RoboDK station: Model of an industrial robot with a technical vision system for palletizing objects in the RoboDK environment.rdk

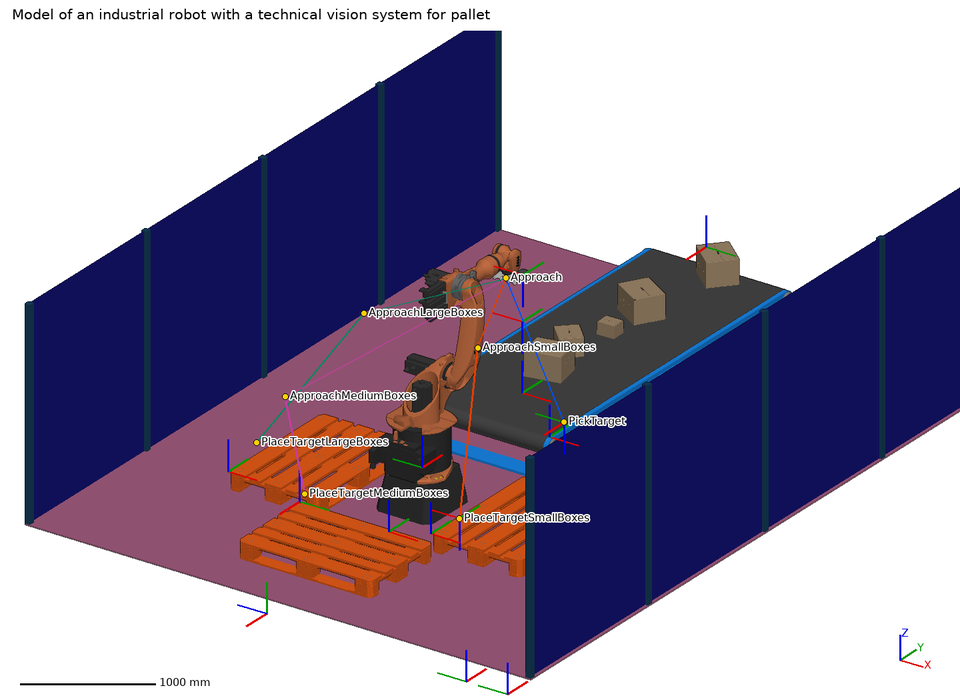
[picture v0: the station drawn from its stored meshes, robots at their saved joint values, targets as dots, program paths as lines]
Station Model of an industrial robot with a technical vision system for palletizing objects in the RoboDK environment (saved by RoboDK 5.9.0). Poses are relative to the parent item; angles as X-Y-Z fixed-axis rotations.
Station parameters (name, value as stored): BOXSPAWNER_SIZE_X, 400.0, BOXSPAWNER_SIZE_Y, 200.0, BOXSPAWNER_SIZE_Z, 200.0, BOXSPAWNER_UNITS, True, BOXSPAWNER_PARENT, Frame 6, BOXSPAWNER_CONV_PARENT, Frame 6, BOXSPAWNER_CONV_MECA, My Mechanism, Box_Dect, No, Box_Num, 9.0, Conveyor_Travel, 400, Box_Height, 0, Box_LengthX, 0, Box_LengthY, 0, RowBoxX, 0, RowBoxY, 0, RowBoxX_Buffer, 0, Pallet_Is_full, 0, IO_5, 1, imageBase64, TestVar, red, TestVar, green, Box_Name, TAGS, ['Add-in', 'Conveying', 'Vision', 'Palletizing', 'HMI'], OPC-UA, opc.tcp://localhost:4840, LIN64
  - frame Vision_Conveyor Base at (600, 1040, 470) mm
    - robot Vision_Conveyor: 1 axes
        modified DH rows (alpha deg, a mm, theta deg, d mm): 0, 0, 0, 0 linear
        base shift (0, 0, 0) mm, rotated rx 90 ry 0 rz 0 deg
        joint limits [-900000] to [900000]; home [0]; saved at [3627]
      - frame Box_Conveyor_Ref at (0, 0, 0) mm
        - object Box 5 at (-4489.76, 220, 612.14) mm, rotated rx -90 ry 10.98 rz 0 deg, size 252 x 305.4 x 216.7 mm, geometry from Box-12x10in-Closed.sld
        - object Box 6 at (-4883.1, 165, 710.16) mm, rotated rx -90 ry -45.22 rz 0 deg, size 189 x 229 x 162.5 mm, geometry from Box-12x10in-Closed.sld
        - object Box 7 at (-5294.47, 110, 625.74) mm, rotated rx -90 ry 1.84 rz 0 deg, size 126 x 152.7 x 108.3 mm, geometry from Box-12x10in-Closed.sld
        - object Box 8 at (-5689.86, 220, 625.52) mm, rotated rx -90 ry -30.95 rz 0 deg, size 252 x 305.4 x 216.7 mm, geometry from Box-12x10in-Closed.sld
        - object Box 9 at (-6510.29, 220, 516.25) mm, rotated rx -90 ry -40.25 rz 0 deg, size 252 x 305.4 x 216.7 mm, geometry from Box-12x10in-Closed.sld
    - frame Box_Init_Ref at (-620, 2900, 220) mm, rotated rx 0 ry 0 rz -90 deg
      - object BoxRef at (0, 0, 0) mm, size 252 x 305.4 x 216.7 mm, geometry from Box-12x10in-Closed.sld
      - object Box 9 at (0, 0, 0) mm, size 252 x 305.4 x 216.7 mm, geometry from Box-12x10in-Closed.sld
    - frame Vision Frame at (-590, 490, 0) mm
      - frame Camera_Frame at (0, 0, 580) mm, rotated rx 180 ry 0 rz 180 deg
    - object Collision Cube at (-1190, -80, -470) mm, size 1200 x 480 x 1200 mm, geometry from Untitled.step
    - target Approach (Cartesian target) at (-668.3, 396.41, 952) mm, rotated rx 180 ry 0 rz -90 deg; joints [0, -77.622, 76.271, 180, -91.351, -90] of KUKA KR 16 3
    - target PickTarget (Cartesian target) at (-42, 249.57, 7) mm, rotated rx 180 ry 0 rz -90 deg; joints [33.97, -27.926, 92.13, 180, -25.796, -56.03] of KUKA KR 16 3
    - frame Frame 15 at (-42.55, 249.57, 7) mm, rotated rx 180 ry 0 rz -90 deg
    - target ApproachSmallBoxes (Cartesian target) at (-168.3, -680, 951.98) mm, rotated rx 180 ry 0 rz -180 deg; joints [90, -128.315, 115.763, 180, -102.552, -90] of KUKA KR 16 3
    - target PlaceTargetSmallBoxes (Cartesian target) at (-18.3, -1130, -221.66) mm, rotated rx 180 ry 0 rz -180 deg; joints [124.695, -10.855, 109.67, 180, 8.815, -55.305] of KUKA KR 16 3
    - frame Frame 16 at (-18.3, -1130, -221.66) mm, rotated rx 180 ry 0 rz -180 deg
    - target ApproachMediumBoxes (Cartesian target) at (-1120, -1790, 729.54) mm, rotated rx 180 ry 0 rz 90 deg; joints [-157.415, -63.979, 77.309, 180, -76.67, -67.415] of KUKA KR 16 3
    - target PlaceTargetMediumBoxes (Cartesian target) at (-1120, -1540, -167.49) mm, rotated rx 180 ry 0 rz 90 deg; joints [-151.77, -16.519, 98.041, 0, 8.479, 118.23] of KUKA KR 16 3
    - target ApproachLargeBoxes (Cartesian target) at (-1190, -680, 951.98) mm, rotated rx 180 ry 0 rz 0 deg; joints [-90, -126.262, 114.986, 180, -101.276, -90] of KUKA KR 16 3
    - target PlaceTargetLargeBoxes (Cartesian target) at (-1840, -1130, -113.32) mm, rotated rx 180 ry 0 rz 0 deg; joints [-111.01, -13.717, 70.817, 180, -32.9, -111.01] of KUKA KR 16 3
  - frame KUKA KR 16 3 Base at (-68.3, 360, 300) mm, rotated rx 0 ry 0 rz 90 deg
    - robot KUKA KR 16 3: 6 axes, payload 16 kg, reach 1611 mm, repeatability 0.05 mm, weight 235 kg
        modified DH rows (alpha deg, a mm, theta deg, d mm): 0, 0, 0, 675; -90, 260, 0, 0; 0, 680, -90, 0; -90, -35, 0, 670; 90, 0, 0, 0; -90, 0, 180, 158
        joint limits [-185, -155, -130, -350, -130, -350] to [185, 35, 154, 350, 130, 350]; home [0, -90, 90, 0, 0, 0]; saved at [0.532, -77.618, 76.266, 180, -91.352, -89.468]
      - tool Vacuum Gripper, TCP at (-10, 0, 40) mm, rotated rx 0 ry 0 rz 90 deg, size 209.9 x 42 x 100 mm
      - frame Camera Reference at (78.3, -93.59, 25.68) mm, rotated rx 0 ry 0 rz 180 deg
        - object SICK VSPP-5F2113 Camera at (0, 0, 0) mm, rotated rx 0 ry 0 rz 90 deg, size 116 x 53 x 38 mm, geometry from SICK-VSPP-5F2113-Camera.sld
    - object Pedestal H500mm (Type 2) at (0, 0, -300) mm, rotated rx 0 ry 0 rz -90 deg, size 506.7 x 560.2 x 300 mm, geometry from Pedestal-H500mm-Type-2.sld
  - frame Pallet at (160, -390, 140) mm
    - frame Pallet_for_small_boxes at (271.7, 150, 0) mm
      - object Pallet 1200x800mm (Transverse) at (0, 0, 0) mm, size 800 x 1200 x 144.2 mm, geometry from Pallet-1200x800mm-Transverse.sld
      - object Box 5 at (0, 0, 0) mm, size 126 x 152.7 x 108.3 mm, geometry from Box_small.sld
    - frame Pallet_for_medium_boxes at (-830, 40, 0) mm, rotated rx 0 ry 0 rz -90 deg
      - object Pallet 1200x800mm (Transverse) at (0, 0, 0) mm, size 800 x 1200 x 144.2 mm, geometry from Pallet-1200x800mm-Transverse.sld
      - object Box 8 at (0, 0, 0) mm, size 189 x 229 x 162.5 mm, geometry from Box_medium.sld
    - frame Pallet_for_large_boxes at (-1550, 150, 0) mm
      - object Pallet 1200x800mm (Transverse) at (0, 0, 0) mm, size 800 x 1200 x 144.2 mm, geometry from Pallet-1200x800mm-Transverse.sld
      - object Box 6 at (0, 0, 0) mm, size 252 x 305.4 x 216.7 mm, geometry from Box_large.sld
  - folder Python
    - Python program Reset_Conveyor (listed below)
    - Python program Delete_Box_Over_The_Edge (listed below)
    - Python program Reset_Tool (listed below)
    - Python program Reset_Pallet (listed below)
    - Python program Conveyor_Advance (listed below)
    - Python program CameraLiveStream (listed below)
    - Python program GeneratePlaceTargetSmallBoxes (listed below)
    - Python program GeneratePlaceTargetMediumBoxes (listed below)
    - Python program GeneratePlaceTargetLargeBoxes (listed below)
    - Python program OpenCV_Parts_Orientation (listed below)
  - folder Other_Programs
    - program DeleteBoxOnEdge (1 instructions, listed below)
    - program PickBox (5 instructions, listed below)
    - program Conveyor_Next (1 instructions, listed below)
    - program DropBoxSmallBoxes (8 instructions, listed below)
    - program DropBoxLargeBoxes (8 instructions, listed below)
    - program PickDropBoxSmallBoxes (2 instructions, listed below)
    - program DropBoxMediumBoxes (8 instructions, listed below)
    - program PickDropBoxMediumBoxes (2 instructions, listed below)
    - program PickDropBoxLargeBoxes (2 instructions, listed below)
    - program Break (1 instructions, listed below)
  - program Reset (4 instructions, listed below)
  - program Main (3 instructions, listed below)
  - frame Shapes at (1890, -1870, -14) mm, rotated rx 0 ry 0 rz 90 deg
    - frame Fence 1 Frame at (0, -370, 0) mm
      - object Fence 1 at (300, 0, 0) mm, size 6050 x 4550 x 1810 mm
  - camera My Camera
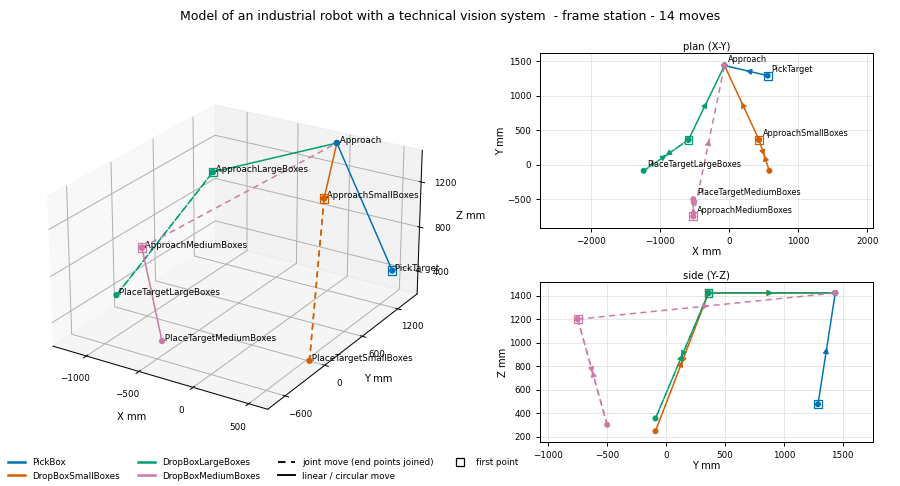
[picture p0: tool path of Model of an industrial robot with a technical vision system for palletizing objects in the RoboDK environment.rdk in frame station, 14 of 14 moves have a stored position in this frame; points joined in program order, loops and branches not executed]

--- Python program Reset_Conveyor ---
# Type help("robolink") or help("robodk") for more information
# Press F5 to run the script
# Documentation: https://robodk.com/doc/en/RoboDK-API.html
# Reference:     https://robodk.com/doc/en/PythonAPI/index.html
# Note: It is not required to keep a copy of this file, your python script is saved with the station
from robodk import robolink
RDK = robolink.Robolink()

#This program reinitialize every mechanisms in the list to position 0
MECHANISM_NAME = "Vision_Conveyor"
REFERENCE_FRAME = "Box_Conveyor_Ref"
#------- Program ------
frame = RDK.Item(REFERENCE_FRAME, robolink.ITEM_TYPE_FRAME)


mechanism = RDK.Item(MECHANISM_NAME,itemtype=robolink.ITEM_TYPE_ROBOT)
if mechanism.Valid():
    mechanism.setJoints([0])


if frame.Valid():
    for item in frame.Childs():
        if item.Type() == robolink.ITEM_TYPE_OBJECT:
            item.Delete()

RDK.setParam("Box_Num", 0)
RDK.setParam("Box_Name", "")
RDK.setParam("Box_X", "")
RDK.setParam("Box_Y", "")
RDK.setParam("Box_Z", "")

RDK.setParam("Box_A", "")
RDK.setParam("Box_B", "")
RDK.setParam("Box_C", "")
RDK.setParam("Box_Name", "")
RDK.setParam("Box_Dect", "No")

--- Python program Delete_Box_Over_The_Edge ---
# Type help("robolink") or help("robodk") for more information
# Press F5 to run the script
# Documentation: https://robodk.com/doc/en/RoboDK-API.html
# Reference:     https://robodk.com/doc/en/PythonAPI/index.html
# Note: It is not required to keep a copy of this file, your python script is saved with the station
from robodk import robolink
RDK = robolink.Robolink()

#This program reinitialize every mechanisms in the list to position 0

REFERENCE_FRAME = "Box_Conveyor_Ref"
COLLISION_CUBE_NAME = "Collision Cube"

#------- Program ------
frame = RDK.Item(REFERENCE_FRAME, robolink.ITEM_TYPE_FRAME)
Collision_Cube = RDK.Item(COLLISION_CUBE_NAME, robolink.ITEM_TYPE_OBJECT)


if frame.Valid():
    for item in frame.Childs():
        if item.Collision(Collision_Cube) or item.IsInside(Collision_Cube):
            if item.Type() == robolink.ITEM_TYPE_OBJECT:
                item.Delete()

--- Python program Reset_Tool ---
# Type help("robolink") or help("robodk") for more information
# Press F5 to run the script
# Documentation: https://robodk.com/doc/en/RoboDK-API.html
# Reference:     https://robodk.com/doc/en/PythonAPI/index.html
# Note: It is not required to keep a copy of this file, your python script is saved with the station
from robodk import robolink
RDK = robolink.Robolink()

#----- CONSTANT -----

TOOL_NAME1 = 'OnRobot VGC10 Vacuum Gripper' #Name of the ref object to copy

#----- PROGRAM -----
tool1 = RDK.Item(TOOL_NAME1,robolink.ITEM_TYPE_TOOL)


if tool1.Valid():
    for item in tool1.Childs():
        if item.Type() == robolink.ITEM_TYPE_OBJECT:
            item.Delete()

--- Python program Reset_Pallet ---
# Type help("robolink") or help("robodk") for more information
# Press F5 to run the script
# Documentation: https://robodk.com/doc/en/RoboDK-API.html
# Reference:     https://robodk.com/doc/en/PythonAPI/index.html
# Note: It is not required to keep a copy of this file, your python script is saved with the station

# You can also use the new version of the API:
from robodk import robolink   # RoboDK API
from robodk import robomath    # Robot toolbox
RDK = robolink.Robolink()

#----- CONSTANT -----

FRAME = 'Pallet' #Name of the ref object to copy
PALLET = "Pallet 1200x800mm (Transverse)"

#----- PROGRAM -----
frame = RDK.Item(FRAME,robolink.ITEM_TYPE_FRAME)


if frame.Valid():
    for item in frame.Childs():
        if item.Type() == robolink.ITEM_TYPE_OBJECT:
            if item.Name() != PALLET:
                item.Delete()


RDK.setParam("RowBoxX",0)
RDK.setParam("RowBoxY",0)
RDK.setParam("RowBoxX_Buffer",0)

--- Python program Conveyor_Advance ---
import random
from robodk import robolink, robomath

RDK = robolink.Robolink()

#----- Constants -----
REFERENCE_FRAME = 'Box_Conveyor_Ref'  # Name of the frame the object will move to
REFERENCE_FRAME_REF = 'Box_Init_Ref'
MECHANISM_NAME = "Vision_Conveyor"

PART_TRAVEL_MM = RDK.getParam("Conveyor_Travel")  # Travel for each box
NEW_REF_OBJECT_NAME = 'BoxRef'  # Name of the ref object to copy
NEW_OBJECT_NAME = 'Box'  # Name of the new object created

# List of predefined sizes for the boxes
BOX_SIZES = [0.5, 0.75, 1.0]

#------- Program ------
frame = RDK.Item(REFERENCE_FRAME, robolink.ITEM_TYPE_FRAME)
frame_ref = RDK.Item(REFERENCE_FRAME_REF, robolink.ITEM_TYPE_FRAME)
ref_obj = RDK.Item(NEW_REF_OBJECT_NAME, robolink.ITEM_TYPE_OBJECT)
mechanism = RDK.Item(MECHANISM_NAME, itemtype=robolink.ITEM_TYPE_ROBOT)

r = random.SystemRandom()

# Randomly choose one of the predefined box sizes
size = r.choice(BOX_SIZES)

x = r.uniform(0, 20)
y = r.uniform(-280, 280)
rotz = r.uniform(-80, 80)

copybox = r.uniform(0, 1)

RDK.setSimulationSpeed(3.5)

if frame.Valid() and ref_obj.Valid() and copybox > 0.1:

    ref_obj.Copy()
    new_obj = RDK.Paste()
    new_obj.setVisible(False)

    boxnum = RDK.getParam("Box_Num")

    RDK.setParam("Box_Num", boxnum + 1)

    new_obj.setName(NEW_OBJECT_NAME + " " + str(int(RDK.getParam("Box_Num"))))
    new_obj.setParent(frame_ref)

    new_obj.setPose(robomath.Offset(new_obj.Pose(), x, y, (frame_ref.Pose()[2, 3] * size) - frame_ref.Pose()[2, 3], 0, 0, rotz))
    new_obj.Scale(size)

    new_obj.setParentStatic(frame)
    new_obj.setVisible(True)
    RDK.Update()

if mechanism.Valid():
    mechanism.MoveJ(mechanism.Joints() + PART_TRAVEL_MM)

--- Python program CameraLiveStream ---
# Type help("robodk.robolink") or help("robodk.robomath") for more information
# Press F5 to run the script
# Documentation: https://robodk.com/doc/en/RoboDK-API.html
# Reference:     https://robodk.com/doc/en/PythonAPI/index.html
#
# This example demonstrates some of the basic functionalities to handle 2D cameras using the RoboDK API for Python.
# It creates/reuses an existing camera, set its parameters, get the image using two different methods and display it to the user as a live stream.
# This is a great starting point for your computer vision algorithms.
#

from robodk import robolink  # RoboDK API
from robodk import robomath  # Robot toolbox
RDK = robolink.Robolink()

# OpenCV is an open source Computer Vision toolkit, which you can use to filter and analyse images
robolink.import_install('cv2', 'opencv-python', RDK)
robolink.import_install('numpy', RDK)
import numpy as np
import cv2 as cv

CAM_NAME = 'My Camera'
CAM_PARAMS = 'SIZE=640x480' # For more options, see https://robodk.com/doc/en/PythonAPI/robodk.html#robodk.robolink.Robolink.Cam2D_Add
WINDOW_NAME = 'My Camera Feed'

#----------------------------------
# Get the camera item
cam_item = RDK.Item(CAM_NAME, robolink.ITEM_TYPE_CAMERA)
if not cam_item.Valid():
    cam_item = RDK.Cam2D_Add(RDK.AddFrame(CAM_NAME + ' Frame'), CAM_PARAMS)
    cam_item.setName(CAM_NAME)
cam_item.setParam('Open', 1)

#----------------------------------
# Create a live feed
while cam_item.setParam('isOpen') == '1':

    #----------------------------------
    # Method 1: Get the camera image, by socket
    img_socket = None
    bytes_img = RDK.Cam2D_Snapshot('', cam_item)
    if isinstance(bytes_img, bytes) and bytes_img != b'':
        nparr = np.frombuffer(bytes_img, np.uint8)
        img_socket = cv.imdecode(nparr, cv.IMREAD_COLOR)
    if img_socket is None:
        break

    #----------------------------------
    # Method 2: Get the camera image, from disk
    img_png = None
    import tempfile
    with tempfile.TemporaryDirectory(prefix='robodk_') as td:
        tf = td + '/temp.png'
        if RDK.Cam2D_Snapshot(tf, cam_item) == 1:
            img_png = cv.imread(tf)
    if img_png is None:
        break

    #----------------------------------
    # Show it to the world!
    cv.imshow(WINDOW_NAME, img_socket)
    key = cv.waitKey(1)
    if key == 27:
        break  # User pressed ESC, exit
    if cv.getWindowProperty(WINDOW_NAME, cv.WND_PROP_VISIBLE) < 1:
        break  # User killed the main window, exit

# Close the preview and the camera. Ensure you call cam_item.setParam('Open', 1) before reusing a camera!
cv.destroyAllWindows()
RDK.Cam2D_Close(cam_item)

--- Python program GeneratePlaceTargetSmallBoxes ---
from robodk.robolink import *  # RoboDK API
from robodk.robomath import *  # Robot toolbox

RDK = Robolink()

PlaceTargetSmallBoxes  = RDK.Item('PlaceTargetSmallBoxes')     # Получение объекта target по имени

position_array = PlaceTargetSmallBoxes.Pose().Pos()             # the same can be applied to targets (taught position)

x_max = 450.000
y_max = -300.000


if position_array[1] < y_max:
    position_array[1] += 300
    PlaceTargetSmallBoxes.setPose(Pose(position_array[0], position_array[1], position_array[2], -180.000, -0.000, 180.000))  # Установите обновленные значения позиции target

elif position_array[0] < x_max:
    position_array[0] += 250
    position_array[1] = -1130.000
    PlaceTargetSmallBoxes.setPose(Pose(position_array[0], position_array[1], position_array[2], -180.000, -0.000, 180.000))  # Установите обновленные значения позиции target

else:
    position_array[0] = -18.297
    position_array[1] = -1130.000
    position_array[2] += 108.341
    PlaceTargetSmallBoxes.setPose(Pose(position_array[0], position_array[1], position_array[2], -180.000, -0.000, 180.000))  # Установите обновленные значения позиции target

# #PlaceTargetSmallBoxes.setPose(Pose(-18.297, -1130.000, -221.659,  -180.000, -0.000, 180.000))

--- Python program GeneratePlaceTargetMediumBoxes ---
from robodk.robolink import *  # RoboDK API
from robodk.robomath import *  # Robot toolbox

RDK = Robolink()

PlaceTargetMediumBoxes  = RDK.Item('PlaceTargetMediumBoxes')     # Получение объекта target по имени
ApproachMediumBoxes  = RDK.Item('ApproachMediumBoxes')

position_array_p = PlaceTargetMediumBoxes.Pose().Pos()             # the same can be applied to targets (taught position)
position_array_a = ApproachMediumBoxes.Pose().Pos()

x_max = -250.000
y_max = -2000.000


if position_array_p[0] < x_max:
    position_array_p[0] += 300
    PlaceTargetMediumBoxes.setPose(Pose(position_array_p[0], position_array_p[1], position_array_p[2], 180.000, -0.000, -90.000))  # Установите обновленные значения позиции target

    position_array_a[0] += 300
    ApproachMediumBoxes.setPose(Pose(position_array_a[0], position_array_a[1], position_array_a[2], 180.000, -0.000, -90.000))

elif position_array_p[1] > y_max:
    position_array_p[0] = -1120.000
    position_array_p[1] -= 250
    PlaceTargetMediumBoxes.setPose(Pose(position_array_p[0], position_array_p[1], position_array_p[2], 180.000, -0.000, -90.000))  # Установите обновленные значения позиции target

    position_array_a[0] = -1120.000
    #position_array_a[1] -= 250
    ApproachMediumBoxes.setPose(Pose(position_array_a[0], position_array_a[1], position_array_a[2], 180.000, -0.000, -90.000))

else:
    position_array_p[0] = -1120.000
    position_array_p[1] = -1540.000
    position_array_p[2] += 162.512
    PlaceTargetMediumBoxes.setPose(Pose(position_array_p[0], position_array_p[1], position_array_p[2], 180.000, -0.000, -90.000))  # Установите обновленные значения позиции target

    position_array_a[0] = -1120.000
    #position_array_a[1] = -1540.000
    ApproachMediumBoxes.setPose(Pose(position_array_a[0], position_array_a[1], position_array_a[2], 180.000, -0.000, -90.000))
# #PlaceTargetMediumBoxes.setPose(Pose(-1120.000, -1540.000, -167.488,  180.000, -0.000, -90.000))

--- Python program GeneratePlaceTargetLargeBoxes ---
from robodk.robolink import *  # RoboDK API
from robodk.robomath import *  # Robot toolbox

RDK = Robolink()

PlaceTargetLargeBoxes  = RDK.Item('PlaceTargetLargeBoxes')     # Получение объекта target по имени

position_array = PlaceTargetLargeBoxes.Pose().Pos()             # the same can be applied to targets (taught position)

x_max = -1300.000
y_max = -350.000


if position_array[1] < y_max:
    position_array[1] += 400
    PlaceTargetLargeBoxes.setPose(Pose(position_array[0], position_array[1], position_array[2],  180.000, 0.000, 0.000))  # Установите обновленные значения позиции target

elif position_array[0] < x_max:
    position_array[0] += 275
    position_array[1] = -1130.000
    PlaceTargetLargeBoxes.setPose(Pose(position_array[0], position_array[1], position_array[2],  180.000, 0.000, 0.000))  # Установите обновленные значения позиции target

else:
    position_array[0] = -1840.000
    position_array[1] = -1130.000
    position_array[2] += 216.683
    PlaceTargetLargeBoxes.setPose(Pose(position_array[0], position_array[1], position_array[2],  180.000, 0.000, 0.000))  # Установите обновленные значения позиции target

# #PlaceTargetLargeBoxes.setPose(Pose(-1840.000, -1130.000, -113.317,  0.000, 0.000, 180.000))
[ -1840.000000, -1130.000000,  -113.317000,     0.000000,     0.000000,   180.000000 ]

--- Python program OpenCV_Parts_Orientation ---
# Type help("robolink") or help("robodk") for more information
# Press F5 to run the script
# Documentation: https://robodk.com/doc/en/RoboDK-API.html
# Reference:     https://robodk.com/doc/en/PythonAPI/index.html
#
# This example shows how to detect the orientation of elongated parts in a camera feed using OpenCV.
# It uses a simulated camera, but it can easily be modified to use an input camera.
# Warning: best results are observe with elongated parts that are symmetrical.
#
# You can find more information in the OpenCV Contours tutorials:
# https://docs.opencv.org/master/d3/d05/tutorial_py_table_of_contents_contours.html

from robodk.robolink import *  # RoboDK API
from robodk.robomath import *  # Robot toolbox

import_install('cv2', 'opencv-contrib-python')
import cv2 as cv
import numpy as np
import matplotlib.pyplot as plt
import math

#----------------------------------
# Settings
PROCESS_COUNT = -1  # How many frames to process before exiting. -1 means indefinitely.

CAM_NAME = "My Camera"

DISPLAY_RESULT = True
WDW_NAME_RESULTS = 'Object detection using the OpenCV library'

DRAW_AXIS_LENGTH = 30

THRESH_MIN = 50
THRESH_MAX = 255
AREA_MIN = 3000
AREA_MAX_SMALL_BOX = 20000
AREA_MIN_MEDIUM_BOX = AREA_MAX_SMALL_BOX
AREA_MAX_MEDIUM_BOX = 40000
AREA_MIN_LARGE_BOX = AREA_MAX_MEDIUM_BOX
AREA_MAX = 70000

Z_SMALL_BOX = 108.341
Z_MEDIUM_BOX = 162.512
Z_LARGE_BOX = 216.683

#----------------------------------
# Get the simulated camera from RoboDK
RDK = Robolink()

PickTarget = RDK.Item('PickTarget')  # Получение объекта target по имени
PickDropBoxSmallBoxes = RDK.Item('PickDropBoxSmallBoxes') # Получите программу DropBoxSmallBoxes по имени
PickDropBoxMediumBoxes = RDK.Item('PickDropBoxMediumBoxes') # Получите программу DropBoxMediumBoxes по имени
PickDropBoxLargeBoxes = RDK.Item('PickDropBoxLargeBoxes') # Получите программу DropBoxLargeBoxes по имени


#PickTarget_pose = target.Pose()  # Получение позиции target

cam_item = RDK.Item(CAM_NAME, ITEM_TYPE_CAMERA)
if not cam_item.Valid():
    raise Exception("Camera not found! %s" % CAM_NAME)
cam_item.setParam('Open', 1)  # Force the camera view to open

#----------------------------------------------
# Create an resizable result window with sliders for parameters
if DISPLAY_RESULT:
    cv.namedWindow(WDW_NAME_RESULTS)

#----------------------------------------------
# Process camera frames
count = 0
while count < PROCESS_COUNT or PROCESS_COUNT < 0:
    count += 1

    #----------------------------------------------
    # Get the image from RoboDK (since 5.3.0)
    bytes_img = RDK.Cam2D_Snapshot("", cam_item)
    if bytes_img == b'':
        raise
    # Image from RoboDK are BGR, uchar, (h,w,3)
    nparr = np.frombuffer(bytes_img, np.uint8)
    img = cv.imdecode(nparr, cv.IMREAD_UNCHANGED)
    if img is None or img.shape == ():
        raise

    #----------------------------------------------
    # The easiest way to extract features is to threshold their intensity with regards to their background
    # Optimal results with light parts on dark background, and vice-versa
    img=cv.bilateralFilter(img,9,75,75)
    hierarchy, img_bw = cv.threshold(cv.cvtColor(img, cv.COLOR_BGR2GRAY), THRESH_MIN, THRESH_MAX, cv.THRESH_BINARY | cv.THRESH_OTSU)

    #----------------------------------------------
    # Find and parse all the contours in the binary image
    contours, hierarchy = cv.findContours(img_bw, cv.RETR_EXTERNAL, cv.CHAIN_APPROX_NONE)
    for i, c in enumerate(contours):
        # Calculate the contour's area
        area = cv.contourArea(c)

        #----------------------------------------------
        # Display the detection to the user (reference image and camera image side by side, with detection results)
        if DISPLAY_RESULT:
            color = (0, 255, 0)

            # Draw the bounding box
            if area > AREA_MIN and area < AREA_MAX:
                rect = cv.minAreaRect(c)
                center = (rect[0][0], rect[0][1])
                width = rect[1][0]
                height = rect[1][1]
                angle = np.radians(rect[2])
                # Angle is [0, 90], and from the horizontal to the bottom left and bottom right edge of the box
                if width < height:
                    angle += math.pi / 2.0
                if angle > math.pi:
                    angle -= math.pi

                box = cv.boxPoints(rect)
                box = np.int0(box)
                cv.drawContours(img, [box], 0, color, 5)

                def rotate(origin, point, angle):
                    """Rotate a point counterclockwise by a given angle (radians) around a given origin."""
                    ox, oy = origin
                    px, py = point
                    qx = ox + math.cos(angle) * (px - ox) - math.sin(angle) * (py - oy)
                    qy = oy + math.sin(angle) * (px - ox) + math.cos(angle) * (py - oy)
                    return qx, qy

                # Construct the Axis parameters
                center_pt = center
                x_axis = (center_pt[0] + DRAW_AXIS_LENGTH, center_pt[1])
                x_axis = rotate(center_pt, x_axis, angle)
                y_axis = rotate(center_pt, x_axis, math.pi / 2.0)

                center_pt = (int(center_pt[0]), int(center_pt[1]))
                x_axis = (int(x_axis[0]), int(x_axis[1]))
                y_axis = (int(y_axis[0]), int(y_axis[1]))



    if area > AREA_MIN and area < AREA_MAX:
        cv.putText(img, f"area: {area}", (10, 30), cv.FONT_HERSHEY_SIMPLEX, 1, (0, 255, 0), 2)
        cv.putText(img, f"x: {center_pt[0]}", (10, 60), cv.FONT_HERSHEY_SIMPLEX, 1, (0, 255, 0), 2)
        cv.putText(img, f"y: {center_pt[1]}", (10, 90), cv.FONT_HERSHEY_SIMPLEX, 1, (0, 255, 0), 2)
        cv.putText(img, f"img.shape: {img.shape}", (10, 120), cv.FONT_HERSHEY_SIMPLEX, 1, (0, 255, 0), 2)

        # Draw the orientation vector
        cv.circle(img, center_pt, 5, (255, 0, 0), -1)
        cv.arrowedLine(img, center_pt, x_axis, (0, 0, 255), 2, cv.LINE_AA)
        cv.arrowedLine(img, center_pt, y_axis, (0, 255, 0), 2, cv.LINE_AA)

        # Draw the angle
        label = '%0.1f' % np.degrees(angle)
        cv.putText(img, label, (center_pt[0] + 30, center_pt[1]), cv.FONT_HERSHEY_SIMPLEX, 0.7, (255, 255, 255), 1, cv.LINE_AA)

        x_delta_small_boxes = center_pt[0] * 972.222 / img.shape[1]
        y_delta_small_boxes = center_pt[1] * 426.554 / img.shape[0]

        x_delta_medium_boxes = center_pt[0] * 910.332 / img.shape[1]
        y_delta_medium_boxes = center_pt[1] * 399.4 / img.shape[0]

        x_delta_large_boxes = center_pt[0] * 848.4434 / img.shape[1]
        y_delta_large_boxes = center_pt[1] * 372.246 / img.shape[0]

        z_rot_delta = np.degrees(angle)
        if z_rot_delta > 90 and z_rot_delta < 180:
            z_rot_delta = z_rot_delta - 180

    cv.imshow(WDW_NAME_RESULTS, img)
    if cv.waitKey(2000) and area > AREA_MIN and area < AREA_MAX:
        break
    else:
        cv.waitKey(1)
        break

    # cv.imshow(WDW_NAME_RESULTS, img)
    # key = cv.waitKey(1)
    # if key == 27:
    #     break  # User pressed ESC, exit
    # if cv.getWindowProperty(WDW_NAME_RESULTS, cv.WND_PROP_VISIBLE) < 1:
    #     break  # User killed the main window, exit

cv.destroyAllWindows()

if area > AREA_MIN and area < AREA_MAX_SMALL_BOX:
    PickTarget.setPose(Pose(-103.889 - x_delta_small_boxes, 276.724 + y_delta_small_boxes, 7.000 + Z_SMALL_BOX,  180.000, -0.000, 90.000 + z_rot_delta)) # Задание позиции target
    PickDropBoxSmallBoxes.RunProgram()     # Запустите программу DropBoxSmallBoxes

if area > AREA_MIN_MEDIUM_BOX and area < AREA_MAX_MEDIUM_BOX:
    PickTarget.setPose(Pose(-134.834 - x_delta_medium_boxes, 290.300 + y_delta_medium_boxes, 7.000 + Z_MEDIUM_BOX,  180.000, -0.000, 90.000 + z_rot_delta)) # Задание позиции target
    PickDropBoxMediumBoxes.RunProgram()     # Запустите программу PickDropBoxMediumBoxes

if area > AREA_MIN_LARGE_BOX and area < AREA_MAX:
    PickTarget.setPose(Pose(-165.779 - x_delta_large_boxes, 303.877 + y_delta_large_boxes, 7.000 + Z_LARGE_BOX,  180.000, -0.000, 90.000 + z_rot_delta)) # Задание позиции target
    PickDropBoxLargeBoxes.RunProgram()     # Запустите программу PickDropBoxLargeBoxes

--- program DeleteBoxOnEdge (robot Vision_Conveyor) ---
  Call Delete_Box_Over_The_Edge

--- program PickBox (robot KUKA KR 16 3) ---
  Set Ref.: Vision_Conveyor Base
  Set Tool: Vacuum Gripper
  MoveL (PickTarget)
  Attach to Vacuum Gripper
  MoveL (Approach)

--- program Conveyor_Next (robot Vision_Conveyor) ---
  Вызов Conveyor_Advance

--- program DropBoxSmallBoxes (robot KUKA KR 16 3) ---
  Set Ref.: Vision_Conveyor Base
  Set Tool: Vacuum Gripper
  MoveL (ApproachSmallBoxes)
  MoveJ (PlaceTargetSmallBoxes)
  Detach from Vacuum Gripper
  MoveJ (ApproachSmallBoxes)
  MoveL (Approach)
  Call GeneratePlaceTargetSmal...: GeneratePlaceTargetSmallBoxes

--- program DropBoxLargeBoxes (robot KUKA KR 16 3) ---
  Set Ref.: Vision_Conveyor Base
  Set Tool: Vacuum Gripper
  MoveL (ApproachLargeBoxes)
  MoveJ (PlaceTargetLargeBoxes)
  Detach from Vacuum Gripper
  MoveJ (ApproachLargeBoxes)
  MoveL (Approach)
  Call GeneratePlaceTargetLarg...: GeneratePlaceTargetLargeBoxes

--- program PickDropBoxSmallBoxes (robot KUKA KR 16 3) ---
  Call PickBox
  Call DropBoxSmallBoxes

--- program DropBoxMediumBoxes (robot KUKA KR 16 3) ---
  Set Ref.: Vision_Conveyor Base
  Set Tool: Vacuum Gripper
  MoveJ (ApproachMediumBoxes)
  MoveJ (PlaceTargetMediumBoxes)
  Detach from Vacuum Gripper
  MoveJ (ApproachMediumBoxes)
  MoveJ (Approach)
  Call GeneratePlaceTargetMedi...: GeneratePlaceTargetMediumBoxes

--- program PickDropBoxMediumBoxes (robot KUKA KR 16 3) ---
  Call PickBox
  Call DropBoxMediumBoxes

--- program PickDropBoxLargeBoxes (robot KUKA KR 16 3) ---
  Call PickBox
  Call DropBoxLargeBoxes

--- program Break (robot KUKA KR 16 3) ---
  Пауза 5.0 s

--- program Reset (robot Vision_Conveyor) ---
  Call Reset_Conveyor
  Call Reset_Tool
  Call Reset_Pallet
  Set Pallet_Is_full=0

--- program Main (robot KUKA KR 16 3) ---
  Call Conveyor_Next
  Вызов Break
  Вызов OpenCV_Parts_Orientation
